// SIMATIC S7-200 SMART project (STEP 7-Micro/WIN SMART), CPU SR40

SYMBOL_TABLE 系统符号
Always_On        SM0.0    // 始终接通
First_Scan_On    SM0.1    // 仅在第一个扫描周期时接通
Clock_1s         SM0.5    // 针对 1 s 的周期时间，时钟脉冲接通 0.5 s，断开 0.5 s.
END_SYMBOL_TABLE

SYMBOL_TABLE 表格 3
延时定时器            T55
报警延时定时器          T56
延时触发             V2.0
报警延时触发           V2.1
液环泵手动            V50.0
罗茨泵手动            V50.1
排污阀手动            V50.2
补液阀手动            V50.3
液环入口阀手动          V50.4
罗茨入口阀手动          V50.5
罗茨液环入口阀手动        V50.6
自动运行模式           V50.7
机组真空值            VD100
入口温度值            VD104
循环温度值            VD108
液位值              VD112
缓冲罐真空值           VD116
调节阀写入            VD120
入口温度报警设定         VD124
入口温度停机设定         VD128
循环温度报警设定         VD132
循环温度停机设定         VD136
低液位报警设定          VD140
高液位报警设定          VD144
目标液位设定           VD148
调节阀中间变量          VD152
罗茨启动真空设定         VD156
罗茨停机真空设定         VD160
目标真空             VD164
调节阀手动设定          VD168
自动步骤             VW20
罗茨频率读取           VW200
罗茨电流读取           VW202
手动频率设定           VW204
频率写入             VW206
频率显示             VW208
电流显示             VW210
故障报警             V300.0
故障急停             V300.1
急停fault          V300.2
流量开关fault        V300.3
罗茨过载fault        V300.4
软起fault          V300.5
变频器fault         V300.6
入口温度过高报警fault    V300.7
入口温度过高急停fault    V301.0
循环温度过高报警fault    V301.1
循环温度过高急停fault    V301.2
液位过高报警fault      V301.3
液位过低报警fault      V301.4
END_SYMBOL_TABLE

ORGANIZATION_BLOCK MAIN:OB1
TITLE=触摸屏通信心跳
BEGIN
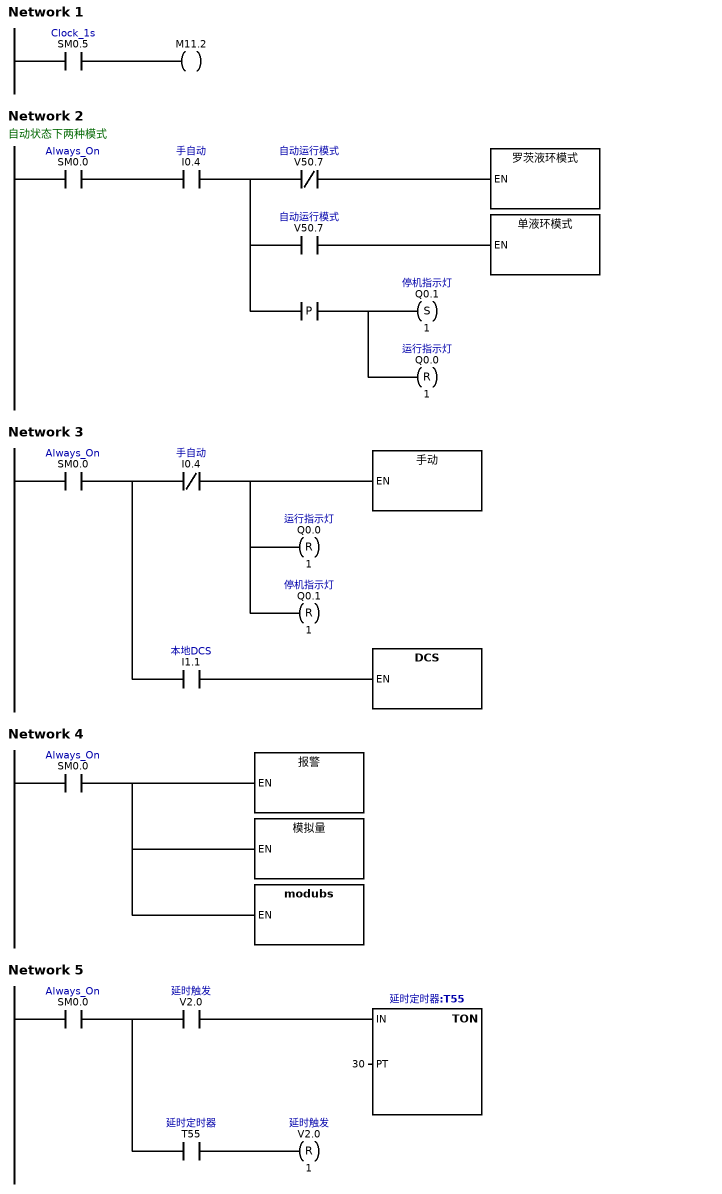
Network 1
LD     Clock_1s:SM0.5
=      M11.2
Network 2
// 自动状态下两种模式
LD     Always_On:SM0.0
A      手自动:I0.4
LPS
AN     自动运行模式:V50.7
CALL   罗茨液环模式:SBR0
LRD
A      自动运行模式:V50.7
CALL   单液环模式:SBR16
LPP
EU
S      停机指示灯:Q0.1, 1
R      运行指示灯:Q0.0, 1
Network 3
LD     Always_On:SM0.0
LPS
AN     手自动:I0.4
CALL   手动:SBR1
R      运行指示灯:Q0.0, 1
R      停机指示灯:Q0.1, 1
LPP
A      本地DCS:I1.1
CALL   DCS:SBR11
Network 4
LD     Always_On:SM0.0
CALL   报警:SBR3
CALL   模拟量:SBR4
CALL   modubs:SBR2
Network 5
LD     Always_On:SM0.0
LPS
A      延时触发:V2.0
TON    延时定时器:T55, 30
LPP
A      延时定时器:T55
R      延时触发:V2.0, 1
END_ORGANIZATION_BLOCK

SUBROUTINE_BLOCK 罗茨液环模式:SBR0
TITLE=
BEGIN
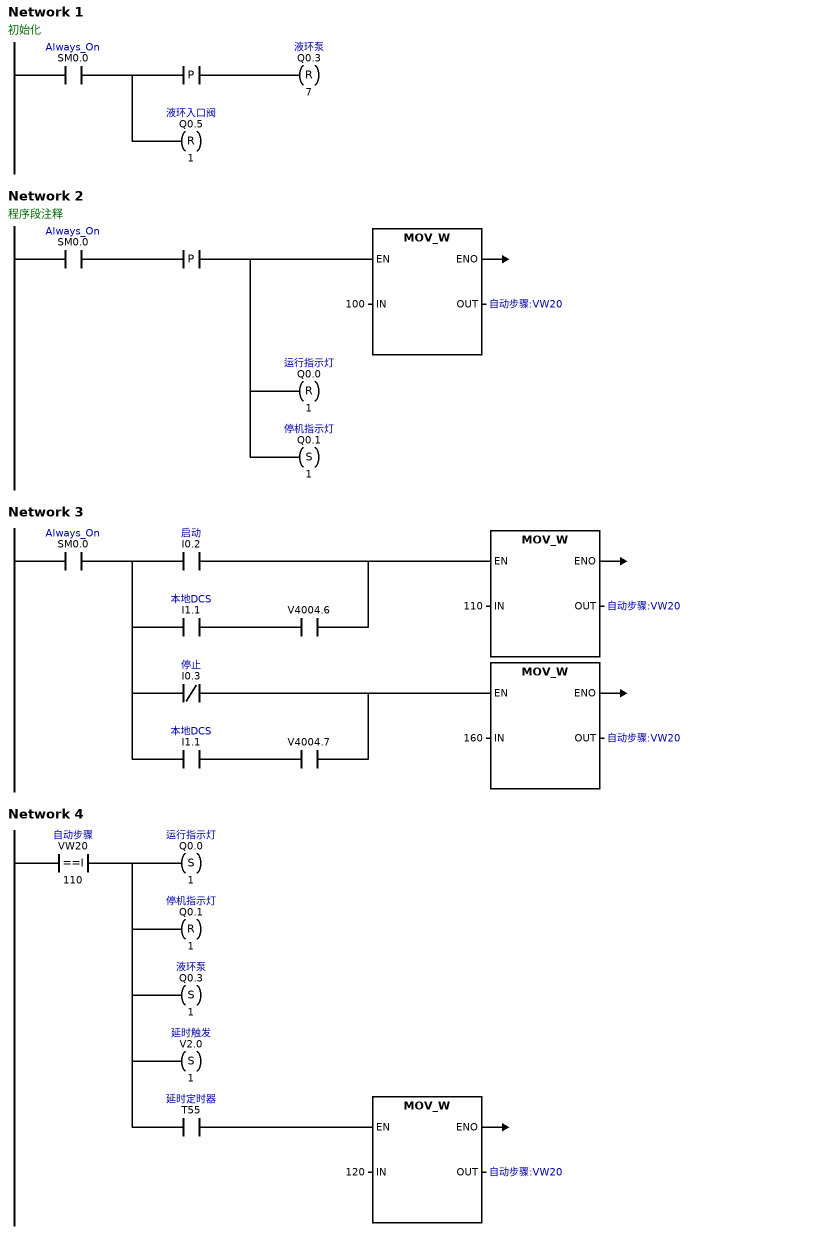
Network 1
// 初始化
LD     Always_On:SM0.0
LPS
EU
R      液环泵:Q0.3, 7
LPP
R      液环入口阀:Q0.5, 1
Network 2
// 程序段注释
LD     Always_On:SM0.0
EU
MOVW   100, 自动步骤:VW20
R      运行指示灯:Q0.0, 1
S      停机指示灯:Q0.1, 1
Network 3
LD     Always_On:SM0.0
LPS
LD     启动:I0.2
LD     本地DCS:I1.1
A      V4004.6
OLD
ALD
MOVW   110, 自动步骤:VW20
LPP
LDN    停止:I0.3
LD     本地DCS:I1.1
A      V4004.7
OLD
ALD
MOVW   160, 自动步骤:VW20
Network 4
LDW=   自动步骤:VW20, 110
S      运行指示灯:Q0.0, 1
R      停机指示灯:Q0.1, 1
S      液环泵:Q0.3, 1
S      延时触发:V2.0, 1
A      延时定时器:T55
MOVW   120, 自动步骤:VW20
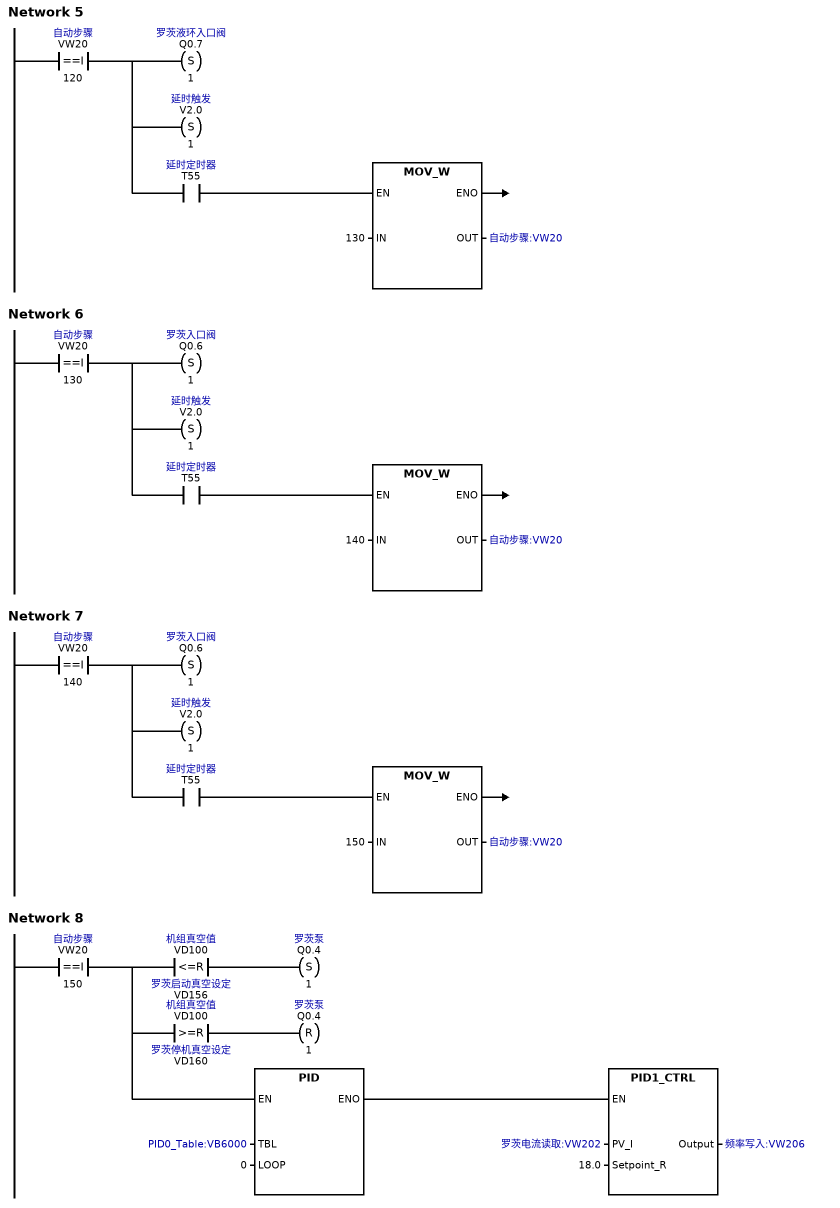
Network 5
LDW=   自动步骤:VW20, 120
S      罗茨液环入口阀:Q0.7, 1
S      延时触发:V2.0, 1
A      延时定时器:T55
MOVW   130, 自动步骤:VW20
Network 6
LDW=   自动步骤:VW20, 130
S      罗茨入口阀:Q0.6, 1
S      延时触发:V2.0, 1
A      延时定时器:T55
MOVW   140, 自动步骤:VW20
Network 7
LDW=   自动步骤:VW20, 140
S      罗茨入口阀:Q0.6, 1
S      延时触发:V2.0, 1
A      延时定时器:T55
MOVW   150, 自动步骤:VW20
Network 8
LDW=   自动步骤:VW20, 150
LPS
AR<=   机组真空值:VD100, 罗茨启动真空设定:VD156
S      罗茨泵:Q0.4, 1
LRD
AR>=   机组真空值:VD100, 罗茨停机真空设定:VD160
R      罗茨泵:Q0.4, 1
LPP
PID    PID0_Table:VB6000, 0
AENO
CALL   PID1_CTRL:SBR10, 罗茨电流读取:VW202, 18.0, 频率写入:VW206
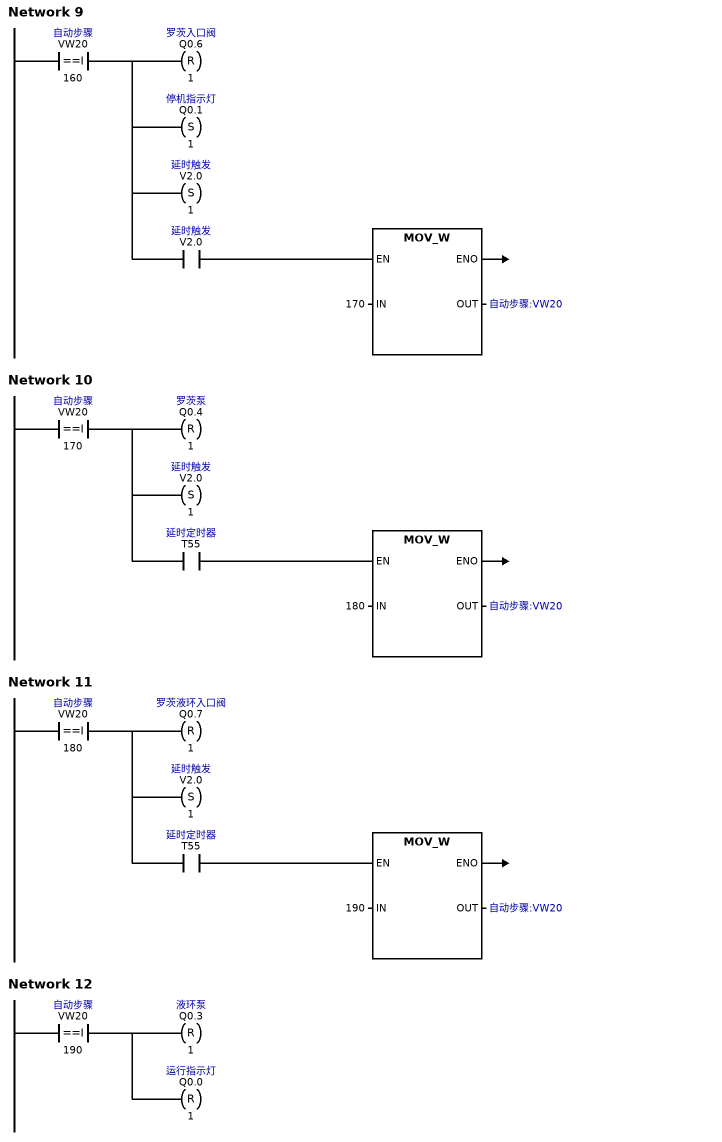
Network 9
LDW=   自动步骤:VW20, 160
R      罗茨入口阀:Q0.6, 1
S      停机指示灯:Q0.1, 1
S      延时触发:V2.0, 1
A      延时触发:V2.0
MOVW   170, 自动步骤:VW20
Network 10
LDW=   自动步骤:VW20, 170
R      罗茨泵:Q0.4, 1
S      延时触发:V2.0, 1
A      延时定时器:T55
MOVW   180, 自动步骤:VW20
Network 11
LDW=   自动步骤:VW20, 180
R      罗茨液环入口阀:Q0.7, 1
S      延时触发:V2.0, 1
A      延时定时器:T55
MOVW   190, 自动步骤:VW20
Network 12
LDW=   自动步骤:VW20, 190
R      液环泵:Q0.3, 1
R      运行指示灯:Q0.0, 1
END_SUBROUTINE_BLOCK

SUBROUTINE_BLOCK 手动:SBR1
TITLE=子程序注释
BEGIN
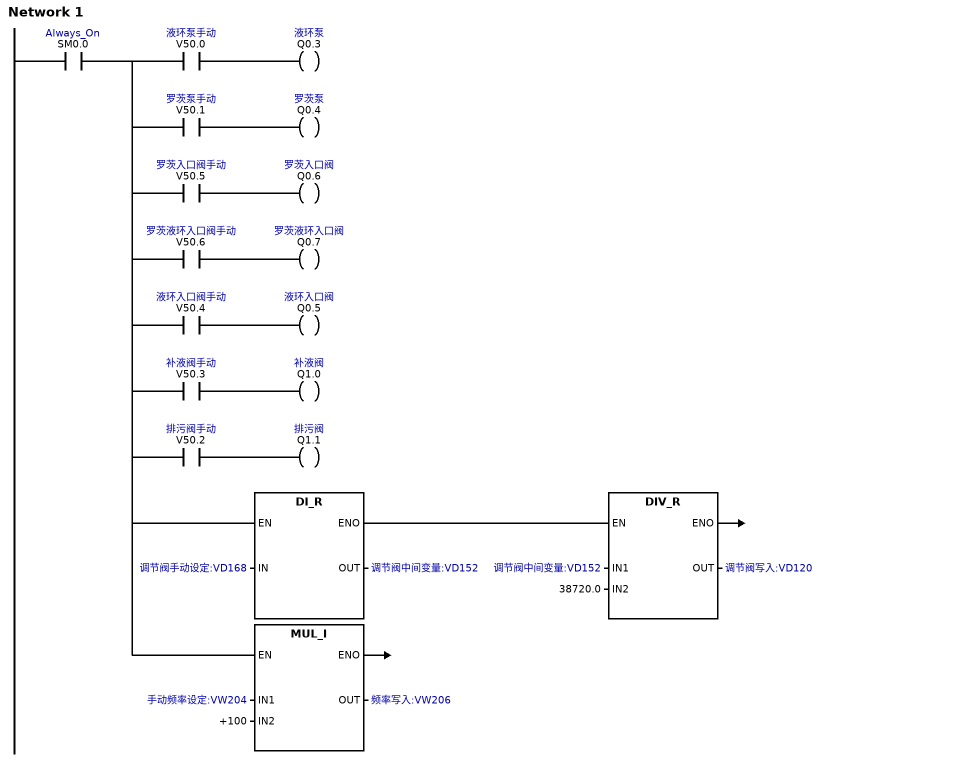
Network 1
LD     Always_On:SM0.0
LPS
A      液环泵手动:V50.0
=      液环泵:Q0.3
LRD
A      罗茨泵手动:V50.1
=      罗茨泵:Q0.4
LRD
A      罗茨入口阀手动:V50.5
=      罗茨入口阀:Q0.6
LRD
A      罗茨液环入口阀手动:V50.6
=      罗茨液环入口阀:Q0.7
LRD
A      液环入口阀手动:V50.4
=      液环入口阀:Q0.5
LRD
A      补液阀手动:V50.3
=      补液阀:Q1.0
LRD
A      排污阀手动:V50.2
=      排污阀:Q1.1
LRD
DTR    调节阀手动设定:VD168, 调节阀中间变量:VD152
AENO
MOVR   调节阀中间变量:VD152, 调节阀写入:VD120
/R     38720.0, 调节阀写入:VD120
LPP
MOVW   手动频率设定:VW204, 频率写入:VW206
*I     +100, 频率写入:VW206
END_SUBROUTINE_BLOCK

SUBROUTINE_BLOCK modubs:SBR2
TITLE=子程序注释
BEGIN
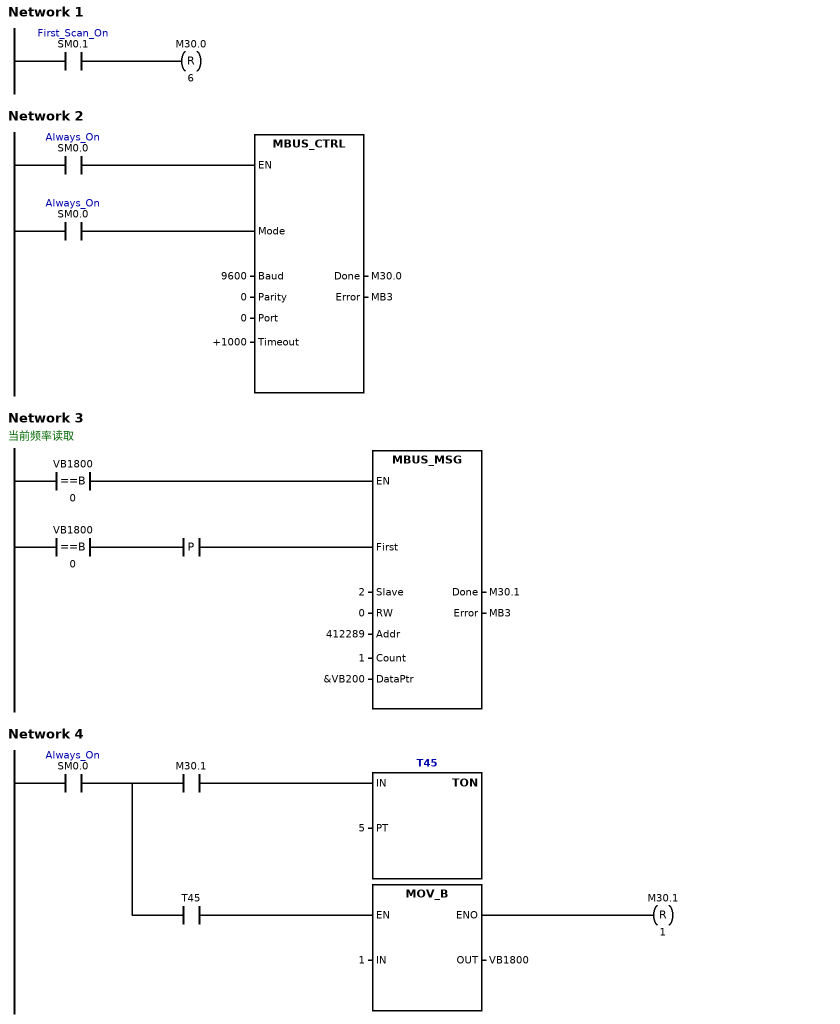
Network 1
LD     First_Scan_On:SM0.1
R      M30.0, 6
Network 2
// 	
LD     Always_On:SM0.0
=      L60.0
LD     Always_On:SM0.0
=      L63.7
LD     L60.0
CALL   MBUS_CTRL:SBR5, L63.7, 9600, 0, 0, +1000, M30.0, MB3
Network 3
// 当前频率读取
LDB=   VB1800, 0
=      L60.0
LDB=   VB1800, 0
EU
=      L63.7
LD     L60.0
CALL   MBUS_MSG:SBR6, L63.7, 2, 0, 412289, 1, &VB200, M30.1, MB3
Network 4
LD     Always_On:SM0.0
LPS
A      M30.1
TON    T45, 5
LPP
A      T45
MOVB   1, VB1800
AENO
R      M30.1, 1
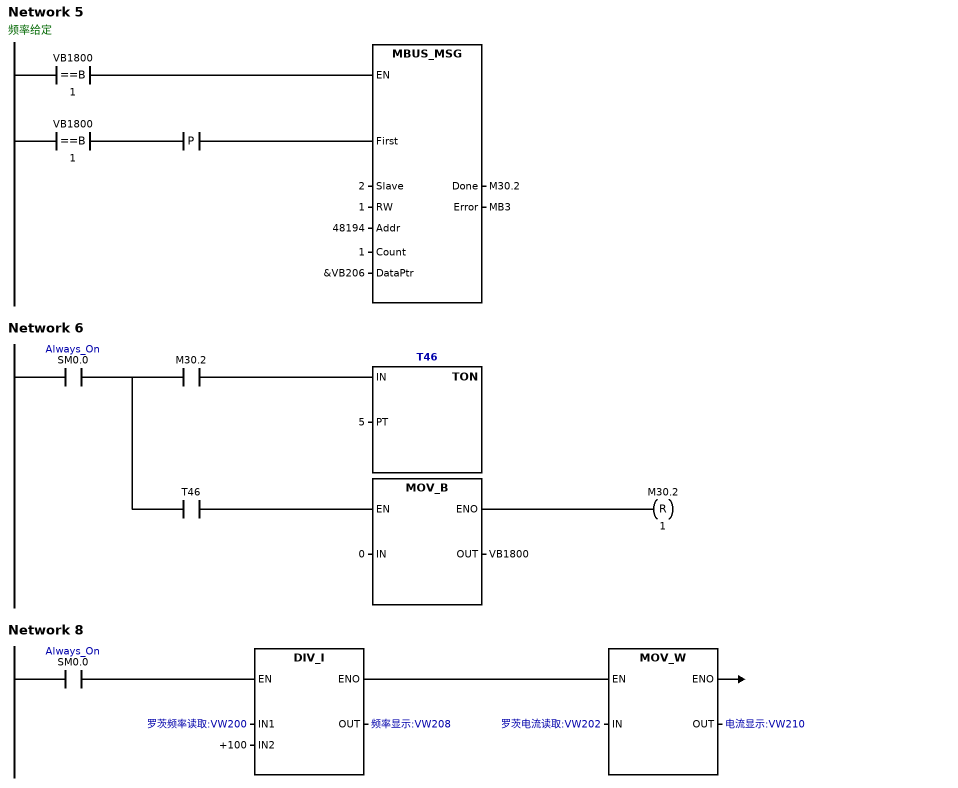
Network 5
// 频率给定
LDB=   VB1800, 1
=      L60.0
LDB=   VB1800, 1
EU
=      L63.7
LD     L60.0
CALL   MBUS_MSG:SBR6, L63.7, 2, 1, 48194, 1, &VB206, M30.2, MB3
Network 6
LD     Always_On:SM0.0
LPS
A      M30.2
TON    T46, 5
LPP
A      T46
MOVB   0, VB1800
AENO
R      M30.2, 1
Network 7
// 电流读取
Network 8
LD     Always_On:SM0.0
MOVW   罗茨频率读取:VW200, 频率显示:VW208
AENO
/I     +100, 频率显示:VW208
AENO
MOVW   罗茨电流读取:VW202, 电流显示:VW210
Network 22
// 程序段注释
END_SUBROUTINE_BLOCK

SUBROUTINE_BLOCK 报警:SBR3
TITLE=子程序注释
BEGIN
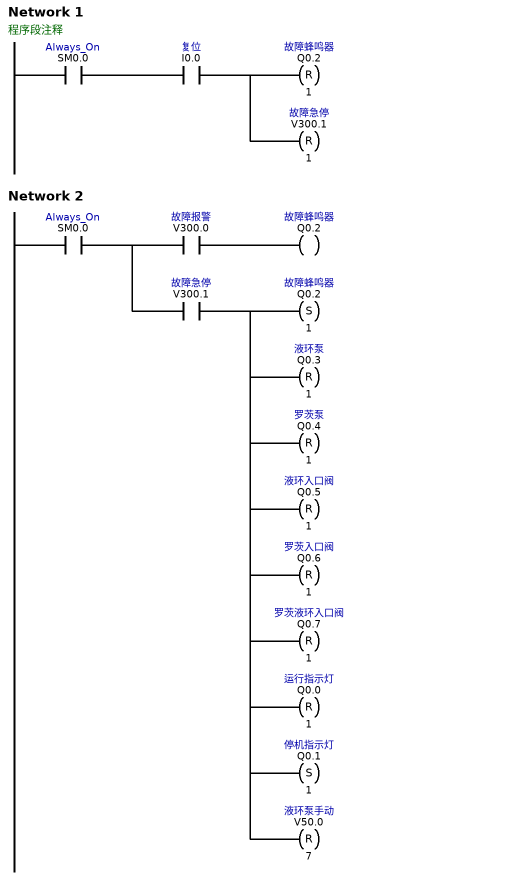
Network 1
// 程序段注释
LD     Always_On:SM0.0
A      复位:I0.0
R      故障蜂鸣器:Q0.2, 1
R      故障急停:V300.1, 1
Network 2
LD     Always_On:SM0.0
LPS
A      故障报警:V300.0
=      故障蜂鸣器:Q0.2
LPP
A      故障急停:V300.1
S      故障蜂鸣器:Q0.2, 1
R      液环泵:Q0.3, 1
R      罗茨泵:Q0.4, 1
R      液环入口阀:Q0.5, 1
R      罗茨入口阀:Q0.6, 1
R      罗茨液环入口阀:Q0.7, 1
R      运行指示灯:Q0.0, 1
S      停机指示灯:Q0.1, 1
R      液环泵手动:V50.0, 7
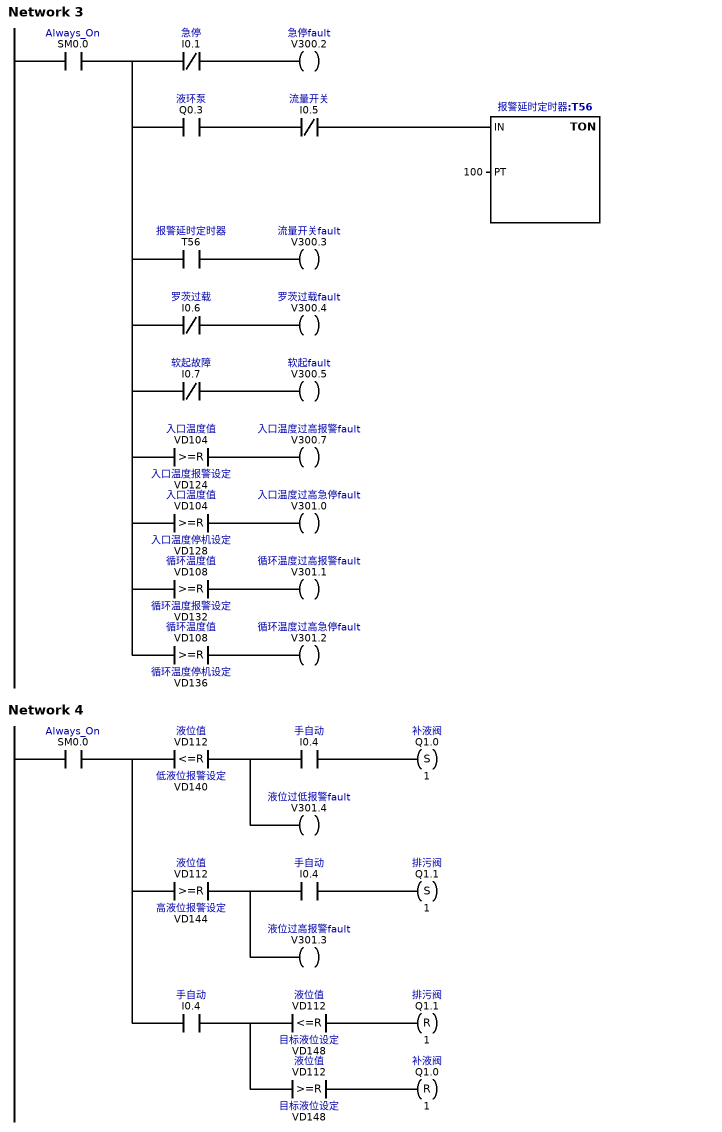
Network 3
LD     Always_On:SM0.0
LPS
AN     急停:I0.1
=      急停fault:V300.2
LRD
A      液环泵:Q0.3
AN     流量开关:I0.5
TON    报警延时定时器:T56, 100
LRD
A      报警延时定时器:T56
=      流量开关fault:V300.3
LRD
AN     罗茨过载:I0.6
=      罗茨过载fault:V300.4
LRD
AN     软起故障:I0.7
=      软起fault:V300.5
LRD
AR>=   入口温度值:VD104, 入口温度报警设定:VD124
=      入口温度过高报警fault:V300.7
LRD
AR>=   入口温度值:VD104, 入口温度停机设定:VD128
=      入口温度过高急停fault:V301.0
LRD
AR>=   循环温度值:VD108, 循环温度报警设定:VD132
=      循环温度过高报警fault:V301.1
LPP
AR>=   循环温度值:VD108, 循环温度停机设定:VD136
=      循环温度过高急停fault:V301.2
Network 4
LD     Always_On:SM0.0
LPS
AR<=   液位值:VD112, 低液位报警设定:VD140
LPS
A      手自动:I0.4
S      补液阀:Q1.0, 1
LPP
=      液位过低报警fault:V301.4
LRD
AR>=   液位值:VD112, 高液位报警设定:VD144
LPS
A      手自动:I0.4
S      排污阀:Q1.1, 1
LPP
=      液位过高报警fault:V301.3
LPP
A      手自动:I0.4
LPS
AR<=   液位值:VD112, 目标液位设定:VD148
R      排污阀:Q1.1, 1
LPP
AR>=   液位值:VD112, 目标液位设定:VD148
R      补液阀:Q1.0, 1
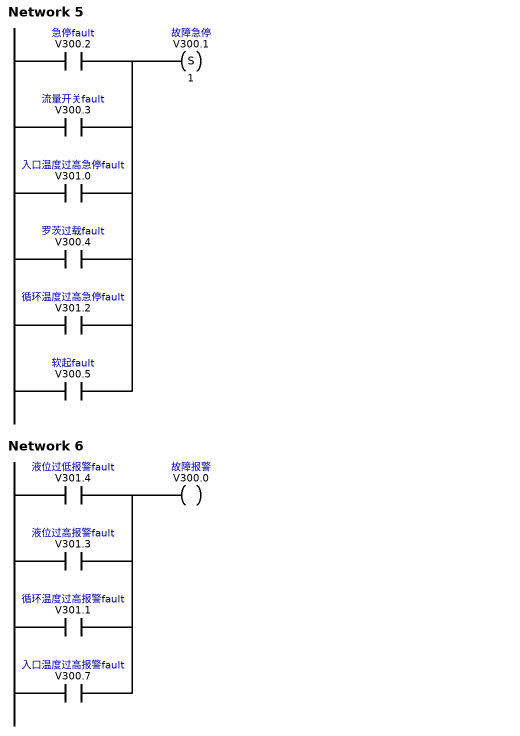
Network 5
LD     急停fault:V300.2
O      流量开关fault:V300.3
O      入口温度过高急停fault:V301.0
O      罗茨过载fault:V300.4
O      循环温度过高急停fault:V301.2
O      软起fault:V300.5
S      故障急停:V300.1, 1
Network 6
LD     液位过低报警fault:V301.4
O      液位过高报警fault:V301.3
O      循环温度过高报警fault:V301.1
O      入口温度过高报警fault:V300.7
=      故障报警:V300.0
END_SUBROUTINE_BLOCK

SUBROUTINE_BLOCK 模拟量:SBR4
TITLE=子程序注释
BEGIN
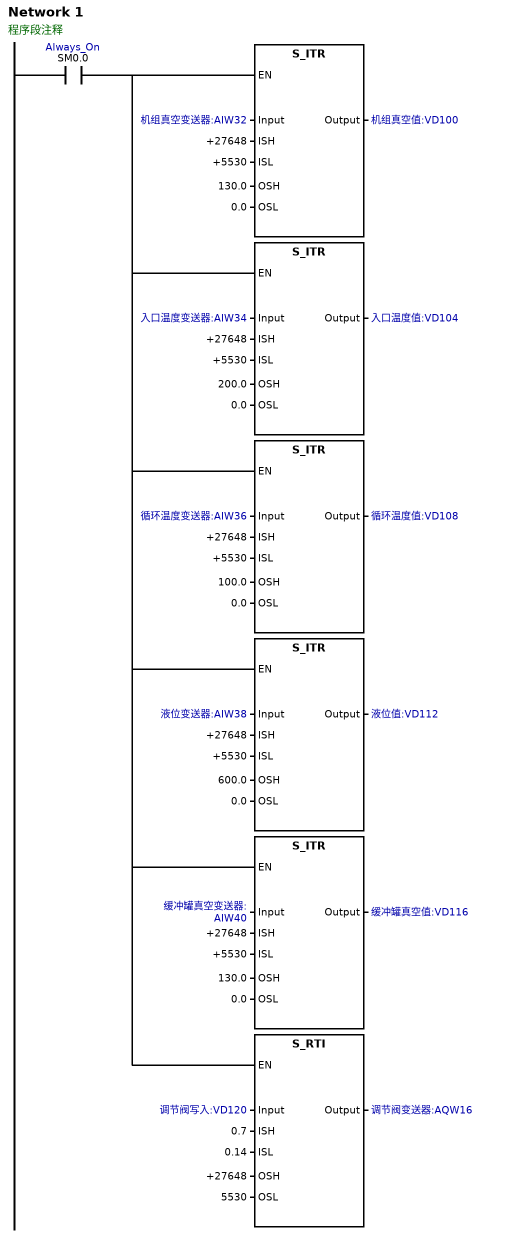
Network 1
// 程序段注释
LD     Always_On:SM0.0
CALL   S_ITR:SBR8, 机组真空变送器:AIW32, +27648, +5530, 130.0, 0.0, 机组真空值:VD100
CALL   S_ITR:SBR8, 入口温度变送器:AIW34, +27648, +5530, 200.0, 0.0, 入口温度值:VD104
CALL   S_ITR:SBR8, 循环温度变送器:AIW36, +27648, +5530, 100.0, 0.0, 循环温度值:VD108
CALL   S_ITR:SBR8, 液位变送器:AIW38, +27648, +5530, 600.0, 0.0, 液位值:VD112
CALL   S_ITR:SBR8, 缓冲罐真空变送器:AIW40, +27648, +5530, 130.0, 0.0, 缓冲罐真空值:VD116
CALL   S_RTI:SBR15, 调节阀写入:VD120, 0.7, 0.14, +27648, 5530, 调节阀变送器:AQW16
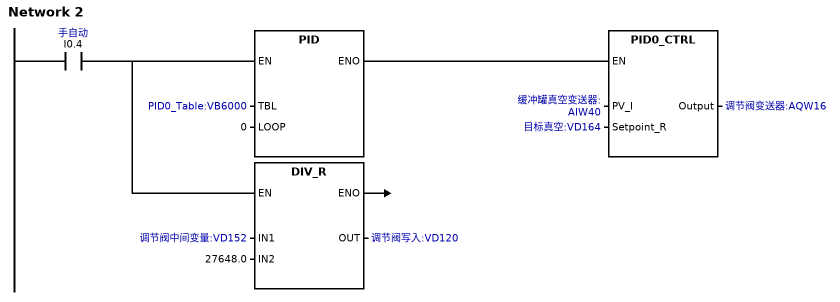
Network 2
LD     手自动:I0.4
LPS
PID    PID0_Table:VB6000, 0
AENO
CALL   PID0_CTRL:SBR9, 缓冲罐真空变送器:AIW40, 目标真空:VD164, 调节阀变送器:AQW16
LPP
MOVR   调节阀中间变量:VD152, 调节阀写入:VD120
/R     27648.0, 调节阀写入:VD120
END_SUBROUTINE_BLOCK

// SBR5: protected block, not included

// SBR6: protected block, not included

// SBR7: protected block, not included

// SBR8: protected block, not included

// SBR9: protected block, not included

// SBR10: protected block, not included

SUBROUTINE_BLOCK DCS:SBR11
TITLE=子程序注释
BEGIN
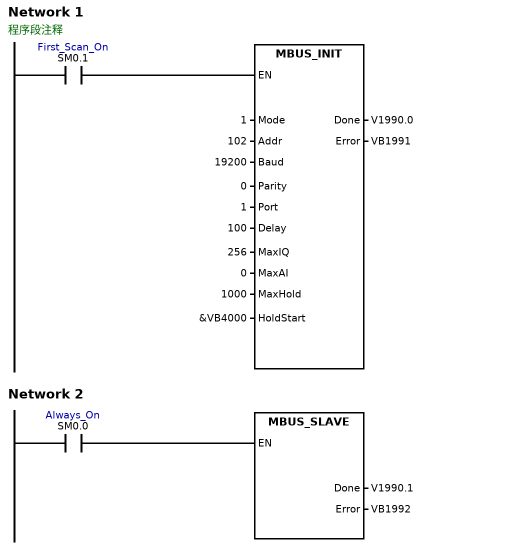
Network 1
// 程序段注释
LD     First_Scan_On:SM0.1
CALL   MBUS_INIT:SBR12, 1, 102, 19200, 0, 1, 100, 256, 0, 1000, &VB4000, V1990.0, VB1991
Network 2
LD     Always_On:SM0.0
CALL   MBUS_SLAVE:SBR13, V1990.1, VB1992
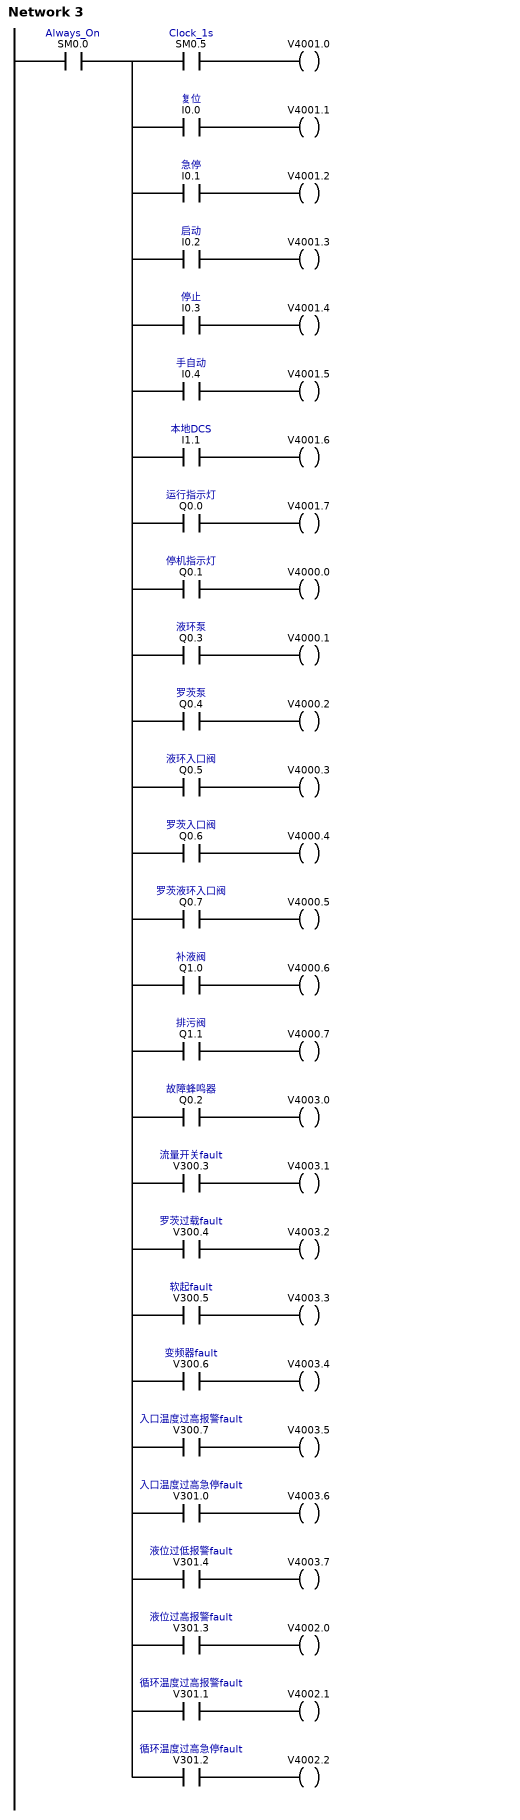
Network 3
LD     Always_On:SM0.0
LPS
A      Clock_1s:SM0.5
=      V4001.0
LRD
A      复位:I0.0
=      V4001.1
LRD
A      急停:I0.1
=      V4001.2
LRD
A      启动:I0.2
=      V4001.3
LRD
A      停止:I0.3
=      V4001.4
LRD
A      手自动:I0.4
=      V4001.5
LRD
A      本地DCS:I1.1
=      V4001.6
LRD
A      运行指示灯:Q0.0
=      V4001.7
LRD
A      停机指示灯:Q0.1
=      V4000.0
LRD
A      液环泵:Q0.3
=      V4000.1
LRD
A      罗茨泵:Q0.4
=      V4000.2
LRD
A      液环入口阀:Q0.5
=      V4000.3
LRD
A      罗茨入口阀:Q0.6
=      V4000.4
LRD
A      罗茨液环入口阀:Q0.7
=      V4000.5
LRD
A      补液阀:Q1.0
=      V4000.6
LRD
A      排污阀:Q1.1
=      V4000.7
LRD
A      故障蜂鸣器:Q0.2
=      V4003.0
LRD
A      流量开关fault:V300.3
=      V4003.1
LRD
A      罗茨过载fault:V300.4
=      V4003.2
LRD
A      软起fault:V300.5
=      V4003.3
LRD
A      变频器fault:V300.6
=      V4003.4
LRD
A      入口温度过高报警fault:V300.7
=      V4003.5
LRD
A      入口温度过高急停fault:V301.0
=      V4003.6
LRD
A      液位过低报警fault:V301.4
=      V4003.7
LRD
A      液位过高报警fault:V301.3
=      V4002.0
LRD
A      循环温度过高报警fault:V301.1
=      V4002.1
LPP
A      循环温度过高急停fault:V301.2
=      V4002.2
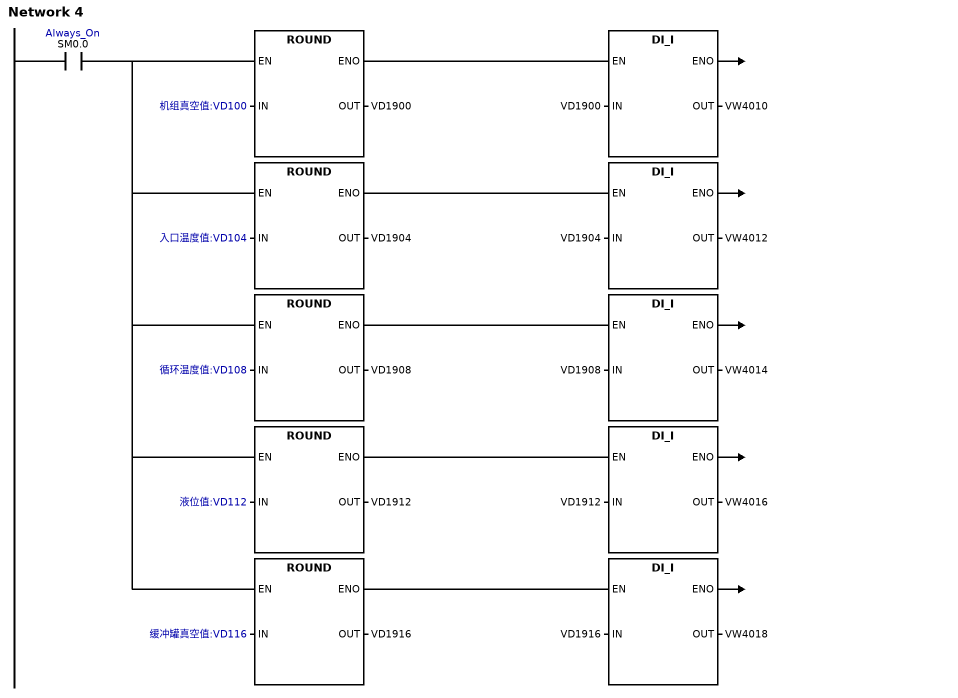
Network 4
LD     Always_On:SM0.0
LPS
ROUND  机组真空值:VD100, VD1900
AENO
DTI    VD1900, VW4010
LRD
ROUND  入口温度值:VD104, VD1904
AENO
DTI    VD1904, VW4012
LRD
ROUND  循环温度值:VD108, VD1908
AENO
DTI    VD1908, VW4014
LRD
ROUND  液位值:VD112, VD1912
AENO
DTI    VD1912, VW4016
LPP
ROUND  缓冲罐真空值:VD116, VD1916
AENO
DTI    VD1916, VW4018
END_SUBROUTINE_BLOCK

// SBR12: protected block, not included

// SBR13: protected block, not included

// SBR14: protected block, not included

// SBR15: protected block, not included

SUBROUTINE_BLOCK 单液环模式:SBR16
TITLE=子程序注释
BEGIN
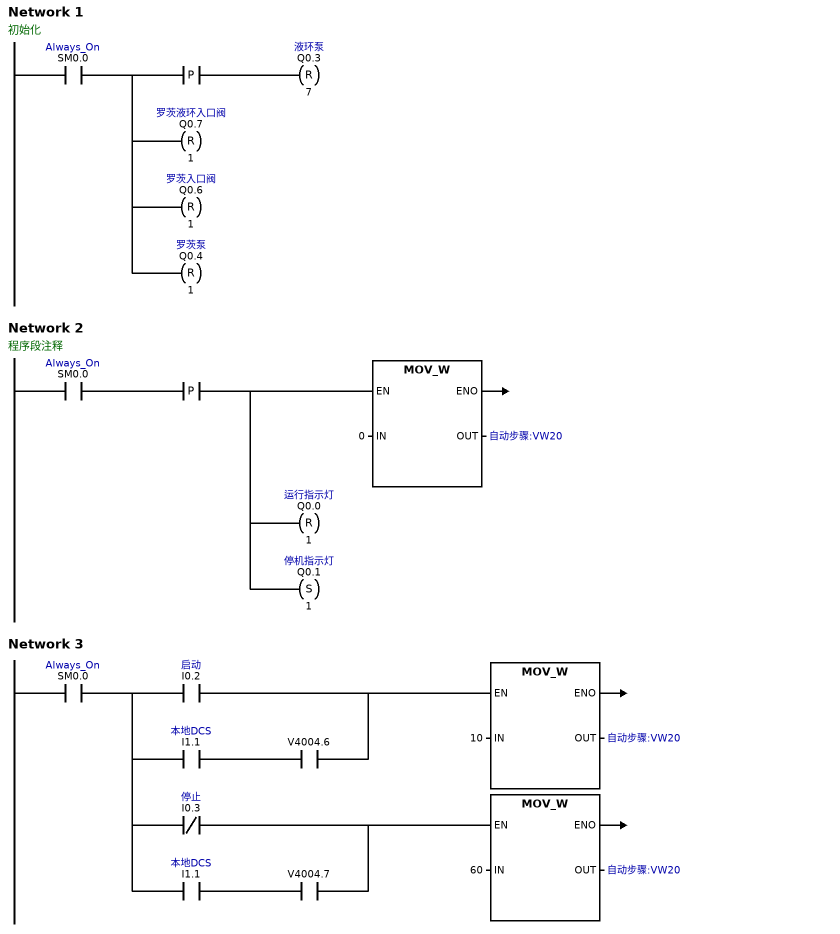
Network 1
// 初始化
LD     Always_On:SM0.0
LPS
EU
R      液环泵:Q0.3, 7
LRD
R      罗茨液环入口阀:Q0.7, 1
LRD
R      罗茨入口阀:Q0.6, 1
LPP
R      罗茨泵:Q0.4, 1
Network 2
// 程序段注释
LD     Always_On:SM0.0
EU
MOVW   0, 自动步骤:VW20
R      运行指示灯:Q0.0, 1
S      停机指示灯:Q0.1, 1
Network 3
LD     Always_On:SM0.0
LPS
LD     启动:I0.2
LD     本地DCS:I1.1
A      V4004.6
OLD
ALD
MOVW   10, 自动步骤:VW20
LPP
LDN    停止:I0.3
LD     本地DCS:I1.1
A      V4004.7
OLD
ALD
MOVW   60, 自动步骤:VW20
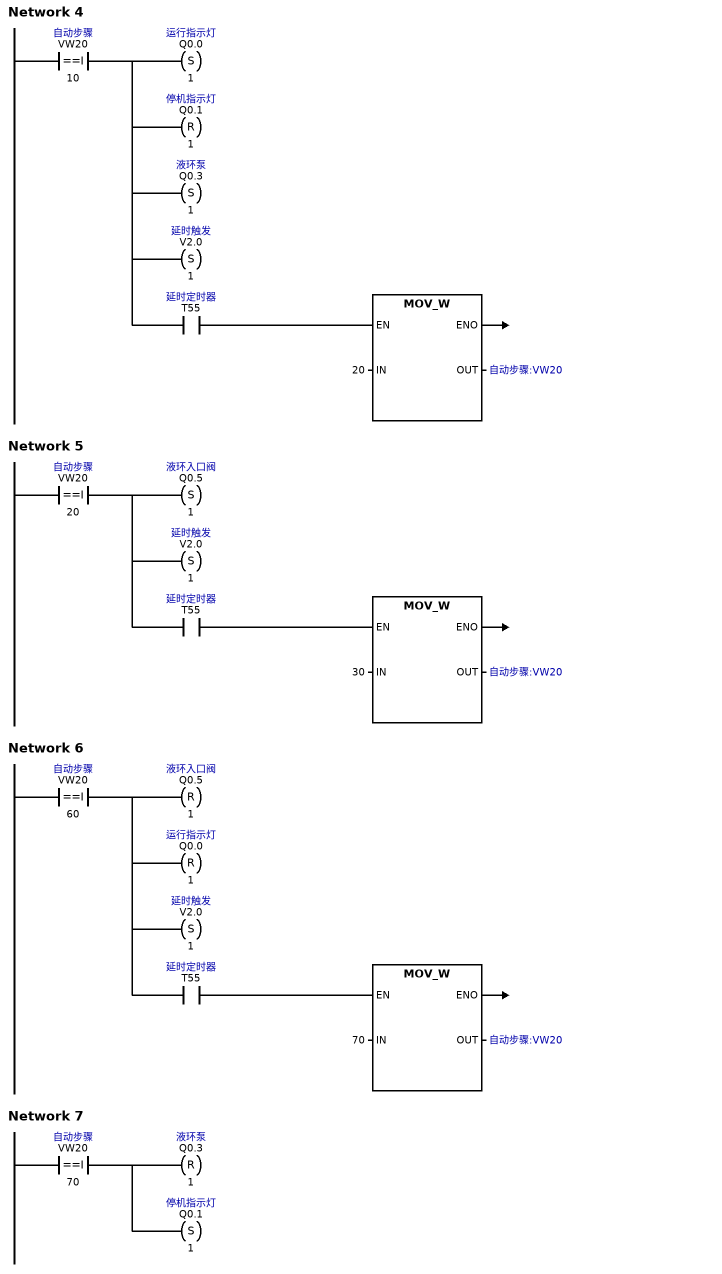
Network 4
LDW=   自动步骤:VW20, 10
S      运行指示灯:Q0.0, 1
R      停机指示灯:Q0.1, 1
S      液环泵:Q0.3, 1
S      延时触发:V2.0, 1
A      延时定时器:T55
MOVW   20, 自动步骤:VW20
Network 5
LDW=   自动步骤:VW20, 20
S      液环入口阀:Q0.5, 1
S      延时触发:V2.0, 1
A      延时定时器:T55
MOVW   30, 自动步骤:VW20
Network 6
LDW=   自动步骤:VW20, 60
R      液环入口阀:Q0.5, 1
R      运行指示灯:Q0.0, 1
S      延时触发:V2.0, 1
A      延时定时器:T55
MOVW   70, 自动步骤:VW20
Network 7
LDW=   自动步骤:VW20, 70
R      液环泵:Q0.3, 1
S      停机指示灯:Q0.1, 1
END_SUBROUTINE_BLOCK
